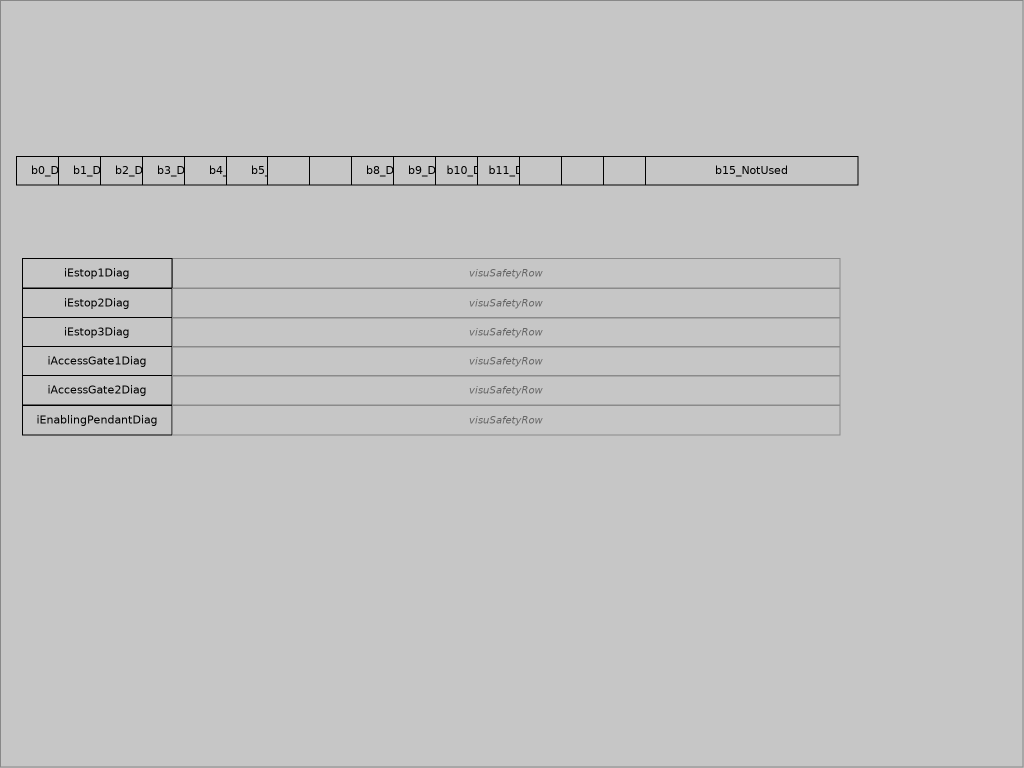
VISUALIZATION Saf_700_SafetyStatus  // 1024x768
    Frame (1068,18 1024x768)
        shows Tmp_000_Template(header := gHMIData.hmiHeader)
    Rectangle (16,156 213x29), angle 45, "b0_DiscrapencyErrorInputGroup1"
    Rectangle (58,156 213x29), angle 45, "b1_DiscrapencyErrorInputGroup2"
    Rectangle (100,156 213x29), angle 45, "b2_DiscrapencyErrorInputGroup3"
    Rectangle (142,156 213x29), angle 45, "b3_DiscrapencyErrorInputGroup4"
    Rectangle (184,156 213x29), angle 45, "b4_EDMmonitoringErrorEDM1"
    Rectangle (226,156 213x29), angle 45, "b5_EDMmonitoringErrorEDM2"
    Rectangle (267,156 213x29), angle 45, "b6_NotUsed"
    Rectangle (309,156 213x29), angle 45, "b7_NotUsed"
    Rectangle (351,156 213x29), angle 45, "b8_DiscrepancyErrorInputGroup1"
    Rectangle (393,156 213x29), angle 45, "b9_DiscrepancyErrorInputGroup2"
    Rectangle (435,156 213x29), angle 45, "b10_DiscrepancyErrorInputGroup3"
    Rectangle (477,156 213x29), angle 45, "b11_DiscrepancyErrorInputGroup4"
    Rectangle (519,156 213x29), angle 45, "b12_NotUsed"
    Rectangle (561,156 213x29), angle 45, "b13_NotUsed"
    Rectangle (603,156 213x29), angle 45, "b14_NotUsed"
    Rectangle (645,156 213x29), angle 45, "b15_NotUsed"
    Frame (172,258 668x30)
        shows visuSafetyRow(dataindi := Safety.iEstop1Diag)
    Rectangle (22,258 150x30), "iEstop1Diag"
    Rectangle (22,288 150x30), "iEstop2Diag"
    Frame (172,288 668x30)
        shows visuSafetyRow(dataindi := Safety.iEstop2Diag)
    Rectangle (22,317 150x30), "iEstop3Diag"
    Frame (172,317 668x30)
        shows visuSafetyRow(dataindi := Safety.iEstop3Diag)
    Rectangle (22,346 150x30), "iAccessGate1Diag"
    Frame (172,346 668x30)
        shows visuSafetyRow(dataindi := Safety.iAccessGate1Diag)
    Rectangle (22,375 150x30), "iAccessGate2Diag"
    Frame (172,375 668x30)
        shows visuSafetyRow(dataindi := Safety.iAccessGate2Diag)
    Rectangle (22,405 150x30), "iEnablingPendantDiag"
    Frame (172,405 668x30)
        shows visuSafetyRow(dataindi := Safety.iEnablingPendantDiag)
END_VISUALIZATION

(* stored: Version 1.1.0.1, ProductVersion 3.1.4024.12
   Visu Saf_700_SafetyStatus: Id {9967be22-951e-4b30-bb9f-541cdbaccc2a} *)
